FUNCTION_BLOCK SymbolProvider
VAR_INPUT
END_VAR
VAR_OUTPUT
END_VAR
VAR
	list : ARRAY[0..99] OF Symbol;
	lastIndex : UINT := 0;
END_VAR

METHOD Get : STRING
VAR_INPUT
	symbol : ANY;
END_VAR
VAR
	i : UINT;
END_VAR
FOR i := 0 TO lastIndex DO
	IF symbol.pValue = list[i].info.pValue THEN
		Get := list[i].description;
		RETURN;
	END_IF
END_FOR
END_METHOD

METHOD Register : BOOL
VAR_INPUT
	symbol				: ANY;
	descriptionName		: STRING;
END_VAR
list[lastIndex].info := symbol;
list[lastIndex].description := descriptionName;
END_METHOD

END_FUNCTION_BLOCK

(* stored: Version 1.1.0.1, ProductVersion 3.1.4024.11
   POU SymbolProvider: Id {ccdf0a92-c83e-4ca8-b12b-f611b2f5fff7}, SpecialFunc None
   Method Get: Id {f9dd9374-6082-4cbf-ab40-385a761477d2}
   Method Register: Id {96c0f692-0f49-4663-ac18-6a8d1a152eb5} *)
